TYPE ST_CameraPoint :
STRUCT
  (*Valus from camera [px/4800dpi]*)
  id                  : UDINT := 0;      (*mark id*)
  x_ref               : DINT := 0;      (*Referenz x deviation [px/4800dpi]*)
  y_ref               : DINT := 0;      (*Referenz y deviation [px/4800dpi]*)
  lx                  : DINT := 0;      (*Referenz in picture x deviation [px/4800dpi]*)
  ly                  : DINT := 0;      (*Referenz in picture y deviation [px/4800dpi]*)
  valid               : BOOL := FALSE;  (*TRUE = PASS, FALSE = FAIL*)
  x                   : DINT := 0;      (*x deviation [px/4800dpi]*)
  y                   : DINT := 0;      (*y deviation [px/4800dpi]*)
END_STRUCT
END_TYPE

(* stored: Version 1.1.0.1, ProductVersion 3.1.4024.3
   DUT ST_CameraPoint: Id {c39ecd96-24fd-4da6-bb67-f1320fea4450} *)
